// TwinCAT 3 PLC project DataTest
// ProgramVersion: 3.1.4024.0
// libraries:
//   Data, * (TomasRompotl)
//   Strings, * (TomasRompotl)
//   Tc2_System, * (Beckhoff Automation GmbH)
//   Tc3_Module, * (Beckhoff Automation GmbH)
//   TcUnit, * (www.tcunit.org)
//   Types, * (TomasRompotl)
// project tree:
//   Comparison/ CompareAnyTypeTest.TcPOU (not stored), ComparisonFunctionsTest.TcPOU (not stored)
//   Manipulate/ ManipulateFunctionsTest.TcPOU
//   / PlcTask.TcTTO (not stored), PRG_Test.TcPOU (not stored), TestTableRow.TcDUT
//   QuickSort/ QuickSortFunctionsTest.TcPOU (not stored)
//   Sort/ SortFunctionsTest.TcPOU (not stored)
//   TableSerialization/ TableDeserializerTest.TcPOU, TableSerializerTest.TcPOU
// (motion and I/O tree: see PLC project typestest)
// real-time tasks:
//   TASK TypesTestTask: cycle T#1ms, priority 20, ADS port 350
//   TASK StringsTestTask: cycle T#1ms, priority 21, ADS port 351
//   TASK DataTestTask: cycle T#1ms, priority 22, ADS port 352
//   TASK MathTestTask: cycle T#1ms, priority 23, ADS port 353
//   TASK TimesTestTask: cycle T#1ms, priority 24, ADS port 354

// ---- TestTableRow.TcDUT
TYPE TestTableRow :
STRUCT
	timestamp : TIME;
	value1 : INT;
	value2 : REAL;
	description : STRING;
END_STRUCT
END_TYPE

// ---- Manipulate/ManipulateFunctionsTest.TcPOU
FUNCTION_BLOCK ManipulateFunctionsTest EXTENDS TcUnit.FB_TestSuite
VAR
END_VAR

ClearDataFunction();
ShiftDataLeftFunction();
ShiftDataRightFunction();
SwapFunction();
SwapByPointerFunction();

METHOD ClearDataFunction : BOOL
VAR
	data : INT;
END_VAR
TcUnit.TEST('Clear data function');

data := 42;
ClearData(data);

AssertEquals_INT(
	Expected := 0,
	Actual := data,
	Message := 'Data memory should be all set to 0');

TEST_FINISHED();
END_METHOD

METHOD ShiftDataLeftFunction : BOOL
VAR
	updatedBuffer : ARRAY[0..LastIndex] OF INT;
	
	expected : ARRAY[0..LastIndex] OF INT;
END_VAR
VAR CONSTANT
	LastIndex : INT := 2;
END_VAR
TcUnit.TEST('Shift data left function');

updatedBuffer[LastIndex] := 1;
ShiftDataLeft(updatedBuffer, SIZEOF(INT));
updatedBuffer[LastIndex] := 2;
ShiftDataLeft(updatedBuffer, SIZEOF(INT));
updatedBuffer[LastIndex] := 3;

expected[0] := 1;
expected[1] := 2;
expected[2] := 3;

AssertArrayEquals_INT(
	Expecteds := expected,
	Actuals := updatedBuffer,
	Message := 'Data should be gradually shifter from end to begin');

TEST_FINISHED();
END_METHOD

METHOD ShiftDataRightFunction : BOOL
VAR
	updatedBuffer : ARRAY[0..LastIndex] OF INT;
	
	expected : ARRAY[0..LastIndex] OF INT;
END_VAR
VAR CONSTANT
	LastIndex : INT := 2;
END_VAR
TcUnit.TEST('Shift data right function');

updatedBuffer[0] := 3;
ShiftDataRight(updatedBuffer, SIZEOF(INT));
updatedBuffer[0] := 2;
ShiftDataRight(updatedBuffer, SIZEOF(INT));
updatedBuffer[0] := 1;

expected[0] := 1;
expected[1] := 2;
expected[2] := 3;

AssertArrayEquals_INT(
	Expecteds := expected,
	Actuals := updatedBuffer,
	Message := 'Data should be gradually shifter from begin to end');

TEST_FINISHED();
END_METHOD

METHOD SwapByPointerFunction : BOOL
VAR
	data1 : INT;
	data2 : INT;
END_VAR
TcUnit.TEST('Swap by pointer function');

data1 := 42;
data2 := 420;

SwapByPointer(ADR(data1), ADR(data2), SIZEOF(data1));

AssertEquals_BOOL(
	Expected := TRUE,
	Actual := data1 = 420 AND data2 = 42,
	Message := 'Data should be swapped');

TEST_FINISHED();
END_METHOD

METHOD SwapFunction : BOOL
VAR
	data1 : INT;
	data2 : INT;
END_VAR
TcUnit.TEST('Swap function');

data1 := 42;
data2 := 420;

Swap(data1, data2);

AssertEquals_BOOL(
	Expected := TRUE,
	Actual := data1 = 420 AND data2 = 42,
	Message := 'Data should be swapped');

TEST_FINISHED();
END_METHOD

END_FUNCTION_BLOCK

// ---- TableSerialization/TableDeserializerTest.TcPOU
FUNCTION_BLOCK TableDeserializerTest EXTENDS TcUnit.FB_TestSuite
VAR
END_VAR

DeserializeTable();
DeserializePartOfTableWithSwappedColumnsAndNoHeader();

METHOD DeserializePartOfTableWithSwappedColumnsAndNoHeader : BOOL
VAR
	data : STRING(1000);
	i : INT;

	table : ARRAY[0..9] OF TestTableRow;
	deserializer : TableDeserializer := (
		DataString := ADR(data)
	);
	
	expected : ARRAY[0..9] OF TestTableRow;
	
	actual : BOOL;
END_VAR
TcUnit.TEST('Deserialize part of table with swapped columns and no header');

// Clear buffers to be able to compare data using memory compare
ClearData(table);
ClearData(expected);

data := 'some text;T#0ms;0,0$Nsome text;T#1ms;3,14$Nsome text;T#2ms;6,28$Nsome text;T#3ms;9,42$Nsome text;T#4ms;12,56$Nsome text;T#5ms;15,700001$Nsome text;T#6ms;18,84$N';

// Define format of data
deserializer.DecimalSeparator := ',';
deserializer.Separator := ';';

// Bind output table
deserializer.DefineRow(table[0]);
deserializer.RowCount := 9;
deserializer.DefineNextColumn(table[0].description);
deserializer.DefineNextColumn(table[0].timestamp);
deserializer.DefineNextColumn(table[0].value2);

// Deserialize
deserializer.Deserialize(includingHeader := FALSE);

// Expected data
FOR i := 0 TO 6 DO
	expected[i].timestamp := TO_TIME(i);
	expected[i].value2 := i * 3.14;
	expected[i].description := 'some text';
END_FOR

actual := TRUE;
FOR i := 0 TO 9 DO
	IF (table[i].timestamp <> expected[i].timestamp
		OR table[i].value1 <> expected[i].value1
		OR ABS(table[i].value2 - expected[i].value2) > 0.1
		OR table[i].description <> expected[i].description) THEN
		
		actual := FALSE;
		EXIT;
	END_IF
END_FOR

AssertEquals_BOOL(
	Expected := TRUE,
	Actual := actual,
	Message := 'Data were not properly deserialized');

TEST_FINISHED();
END_METHOD

METHOD DeserializeTable : BOOL
VAR
	data : STRING(1000);
	i : INT;

	columnNames : ARRAY[0..3] OF T_MaxString;
	table : ARRAY[0..9] OF TestTableRow;
	deserializer : TableDeserializer := (
		DataString := ADR(data)
	);
	
	expected : ARRAY[0..9] OF TestTableRow;
	expectedHeader : ARRAY[0..3] OF T_MaxString;
	
	actual : BOOL;
END_VAR
TcUnit.TEST('Deserialize table');

// Clear buffers to be able to compare data using memory compare
ClearData(columnNames);
ClearData(table);
ClearData(expectedHeader);
ClearData(expected);

data := 'Timestamp;Value 1;Value 2;Description$NT#0ms;0;0,0;some text$NT#1ms;1;3,14;some text$NT#2ms;2;6,28;some text$NT#3ms;3;9,42;some text$NT#4ms;4;12,56;some text$NT#5ms;5;15,700001;some text$NT#6ms;6;18,84;some text$NT#7ms;7;21,98;some text$NT#8ms;8;25,12;some text$NT#9ms;9;28,26;some text';

// Define format of data
deserializer.DecimalSeparator := ',';
deserializer.Separator := ';';

// Bind output table
deserializer.DefineRow(table[0]);
deserializer.RowCount := 10;
deserializer.DefineNextColumn(table[0].timestamp);
deserializer.DefineNextColumn(table[0].value1);
deserializer.DefineNextColumn(table[0].value2);
deserializer.DefineNextColumn(table[0].description);
deserializer.DefineColumnNamesOutput(columnNames);

// Deserialize
deserializer.Deserialize(includingHeader := TRUE);

// Expected data
expectedHeader[0] := 'Timestamp';
expectedHeader[1] := 'Value 1';
expectedHeader[2] := 'Value 2';
expectedHeader[3] := 'Description';
FOR i := 0 TO 9 DO
	expected[i].timestamp := TO_TIME(i);
	expected[i].value1 := i;
	expected[i].value2 := i * 3.14;
	expected[i].description := 'some text';
END_FOR

actual := TRUE;
FOR i := 0 TO 9 DO
	IF (table[i].timestamp <> expected[i].timestamp
		OR table[i].value1 <> expected[i].value1
		OR ABS(table[i].value2 - expected[i].value2) > 0.1
		OR table[i].description <> expected[i].description) THEN
		
		actual := FALSE;
		EXIT;
	END_IF
END_FOR

AssertEquals_BOOL(
	Expected := TRUE,
	Actual := MEMCMP(ADR(columnNames), ADR(expectedHeader), SIZEOF(columnNames)) = 0,
	Message := 'Header was not properly deserialized');
	
AssertEquals_BOOL(
	Expected := TRUE,
	Actual := actual,
	Message := 'Data were not properly deserialized');

TEST_FINISHED();
END_METHOD

END_FUNCTION_BLOCK

// ---- TableSerialization/TableSerializerTest.TcPOU
FUNCTION_BLOCK TableSerializerTest EXTENDS TcUnit.FB_TestSuite
VAR
END_VAR

SerializeTable();
SerializePartOfTableAndSwapColumnsAndWithoutHeader();

METHOD SerializePartOfTableAndSwapColumnsAndWithoutHeader : BOOL
VAR
	table : ARRAY[0..9] OF TestTableRow;
	i : INT;
	
	buffer : STRING(1000);
	sb : StringBuilderExtBuffer := (Buffer := ToAnyType(buffer));
	serializer : TableSerializer := (
		StringBuilder := sb
	);
	
	expected : STRING(1000);
END_VAR
TcUnit.TEST('Serialize part of table and swap columns');

// Prepare data
FOR i := 0 TO 9 DO
	table[i].timestamp := TO_TIME(i);
	table[i].value1 := i;
	table[i].value2 := i * 3.14;
	table[i].description := 'some text';
END_FOR

// Setup serialization
serializer.DecimalSeparator := ',';
serializer.Separator := ';';

// Bind data
serializer.DefineRow(table[0]);
serializer.RowCount := 7;
// Column order is different than structure
serializer.DefineNextColumn(table[0].description);
serializer.DefineNextColumn(table[0].timestamp);
serializer.DefineNextColumn(table[0].value2);

// Serialize
serializer.Serialize(includeHeader := FALSE, clearBuffer := TRUE);

expected := 'some text;T#0ms;0,0$Nsome text;T#1ms;3,14$Nsome text;T#2ms;6,28$Nsome text;T#3ms;9,42$Nsome text;T#4ms;12,56$Nsome text;T#5ms;15,700001$Nsome text;T#6ms;18,84';

AssertEquals_BOOL(
	Expected := TRUE,
	Actual := expected = buffer,
	Message := 'Table was not properly serialized');

TEST_FINISHED();
END_METHOD

METHOD SerializeTable : BOOL
VAR
	table : ARRAY[0..9] OF TestTableRow;
	i : INT;
	
	buffer : STRING(1000);
	sb : StringBuilderExtBuffer := (Buffer := ToAnyType(buffer));
	serializer : TableSerializer := (
		StringBuilder := sb
	);
	
	expected : STRING(1000);
END_VAR
TcUnit.TEST('Serialize table');

// Prepare data
FOR i := 0 TO 9 DO
	table[i].timestamp := TO_TIME(i);
	table[i].value1 := i;
	table[i].value2 := i * 3.14;
	table[i].description := 'some text';
END_FOR

// Setup serialization
serializer.DecimalSeparator := ',';
serializer.Separator := ';';

// Bind data
serializer.DefineRow(table[0]);
serializer.RowCount := 10;
serializer.DefineNextColumnWithName(table[0].timestamp, 'Timestamp');
serializer.DefineNextColumnWithName(table[0].value1, 'Value 1');
serializer.DefineNextColumnWithName(table[0].value2, 'Value 2');
serializer.DefineNextColumnWithName(table[0].description, 'Description');

// Serialize
serializer.Serialize(includeHeader := TRUE, clearBuffer := TRUE);

expected := 'Timestamp;Value 1;Value 2;Description$NT#0ms;0;0,0;some text$NT#1ms;1;3,14;some text$NT#2ms;2;6,28;some text$NT#3ms;3;9,42;some text$NT#4ms;4;12,56;some text$NT#5ms;5;15,700001;some text$NT#6ms;6;18,84;some text$NT#7ms;7;21,98;some text$NT#8ms;8;25,12;some text$NT#9ms;9;28,26;some text';

AssertEquals_BOOL(
	Expected := TRUE,
	Actual := expected = buffer,
	Message := 'Table was not properly serialized');

TEST_FINISHED();
END_METHOD

END_FUNCTION_BLOCK
